FUNCTION_BLOCK XtsMoverManager
VAR_INPUT
END_VAR
VAR_OUTPUT
END_VAR
VAR
END_VAR

END_FUNCTION_BLOCK

(* stored: Version 1.1.0.1, ProductVersion 3.1.4024.6
   POU XtsMoverManager: Id {4b45940e-4817-4260-a891-e07dd3ca95d8}, SpecialFunc None *)
